PROGRAM PRG_Log
VAR
END_VAR

//-----------------------------------------------------------------------------------------
//
//                  				PRG_Log
//
//								Gestion des Log     			
//-----------------------------------------------------------------------------------------
//
//Auteur: G.GOETZ (inspired by S.MANTZER)
//Création: 04.02.2026
//Dernière modification : 04.02.2026 (G.GOETZ)
//       			
//-----------------------------------------------------------------------------------------
//
//     							Liste des modifications  	
//
// 04.02.2026 (G.GOETZ) -> Création		
//-----------------------------------------------------------------------------------------

(** LOG WM **)
	PRG_LOG_WM();

END_PROGRAM

(* stored: Version 1.1.0.1, ProductVersion 3.1.4026.17
   POU PRG_Log: Id {be287b8d-6d84-4fd2-aa5c-09d38f9aeab7}, SpecialFunc None *)
